FUNCTION_BLOCK earth_fault_1_2 (* Composite Function Block Type *)
  (* Standard: 61499-2 *)
  (* Version 0.0, 3/23/2016, gulzha, nxtControl GmbH, template *)
  PACKAGE Main;
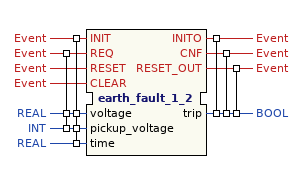
  EVENT_INPUT
    INIT WITH pickup_voltage, voltage, time; (* Initialization Request *)
    REQ WITH pickup_voltage, voltage; (* Normal Execution Request *)
    RESET;
    CLEAR;
  END_EVENT
  EVENT_OUTPUT
    INITO WITH trip; (* Initialization Confirm *)
    CNF WITH trip; (* Execution Confirmation *)
    RESET_OUT WITH trip;
  END_EVENT
  VAR_INPUT
    voltage : REAL;
    pickup_voltage : INT;
    time : REAL;
  END_VAR
  VAR_OUTPUT
    trip : BOOL;
  END_VAR
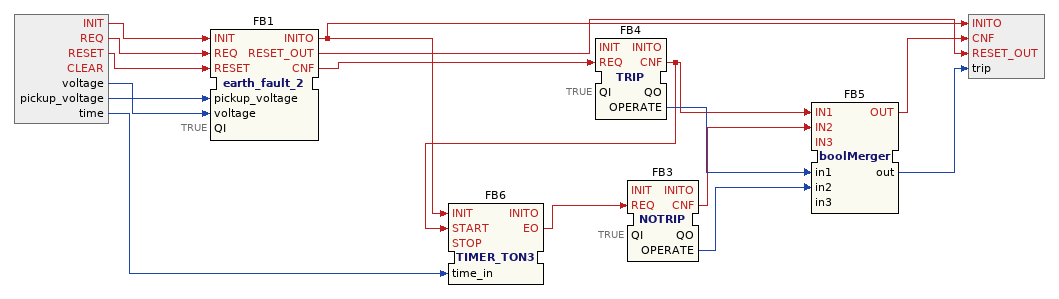
  FBS
    FB1 : earth_fault_2(QI := TRUE);
    FB3 : NOTRIP(QI := TRUE);
    FB4 : TRIP(QI := TRUE);
    FB5 : boolMerger;
    FB6 : TIMER_TON3;
  END_FBS
  EVENT_CONNECTIONS
    INIT TO FB1.INIT;
    FB1.INITO TO INITO;
    REQ TO FB1.REQ;
    RESET TO FB1.RESET;
    FB1.RESET_OUT TO RESET_OUT;
    FB1.CNF TO FB4.REQ;
    FB4.CNF TO FB6.START;
    FB4.CNF TO FB5.IN1;
    FB3.CNF TO FB5.IN2;
    FB5.OUT TO CNF;
    FB6.EO TO FB3.REQ;
    FB1.INITO TO FB6.INIT;
  END_CONNECTIONS
  DATA_CONNECTIONS
    pickup_voltage TO FB1.pickup_voltage;
    voltage TO FB1.voltage;
    FB4.OPERATE TO FB5.in1;
    FB3.OPERATE TO FB5.in2;
    FB5.out TO trip;
    time TO FB6.time_in;
  END_CONNECTIONS
END_FUNCTION_BLOCK
